PROGRAM Clock_2Sec_refresh_
VAR
	timer:INT;
END_VAR

timer:=timer+1;
IF timer=4 THEN
	timer:=0;
END_IF
IF timer < 2 THEN
	HMI_blink_2:=TRUE;
ELSE 
	HMI_blink_2:=FALSE;
END_IF

END_PROGRAM

(* stored: Version 1.1.0.1, ProductVersion 3.1.4022.18
   POU Clock_2Sec_refresh_: Id {56e45688-2d72-4592-86cd-5aed819ea41a}, SpecialFunc None *)
